// TIA Portal V19 export
FUNCTION "@LOAD CALCULATE" : Void   // FC20, LAD
{ S7_Optimized_Access := 'TRUE' }
// stored: SetENOAutomatically false
   VAR_INPUT
      "MFG PROCESS BUFF" : Int;
      "MATERIAL SUCTION BUFF" : Int;
      "MOVE PV" : Real;
      PV : Real;
   END_VAR
   VAR_OUTPUT
      "PURIFIED CALCULATE PV" : Real;
      "MATERIAL SORBITOL CALCULATE PV" : Real;
      "MATERIAL GLUCOSE CALCULATE PV" : Real;
      "MATERIAL SUCTION CALCULATE PV" : Real;
   END_VAR
BEGIN

REGION Network 1
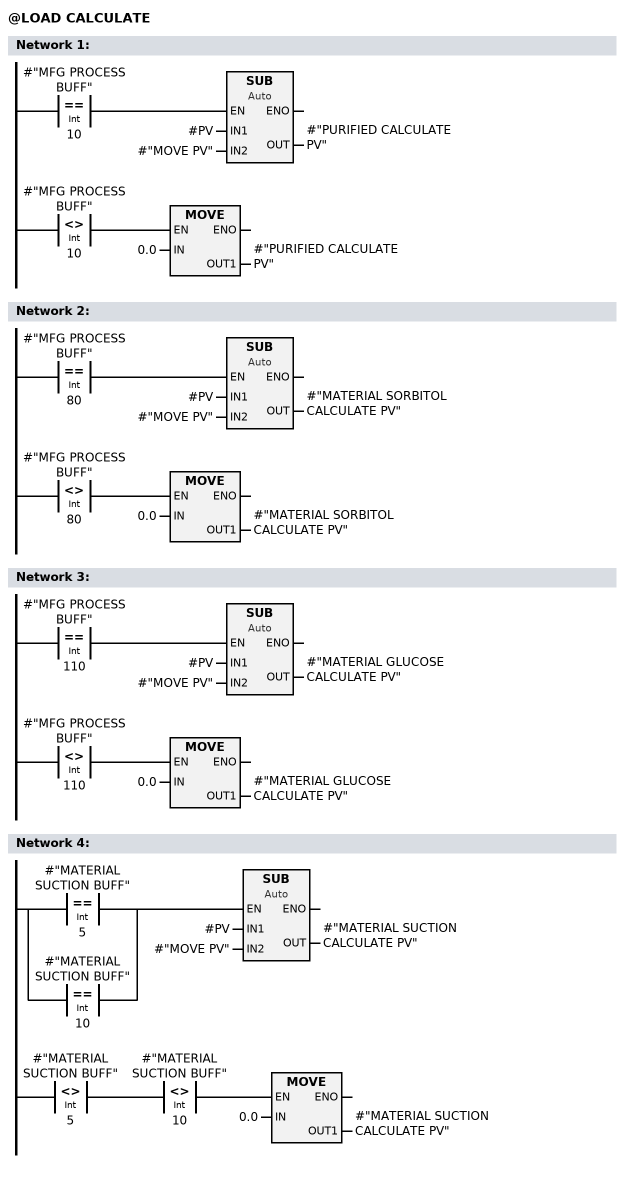
   RUNG wire#powerrail
      { S7_Templates := "SrcType := Int" } EQ_Contact(in1 := #"MFG PROCESS BUFF", in2 := 10)
      Sub(in1 := #PV, in2 := #"MOVE PV", out => #"PURIFIED CALCULATE PV")
   END_RUNG
   RUNG wire#powerrail
      { S7_Templates := "SrcType := Int" } NE_Contact(in1 := #"MFG PROCESS BUFF", in2 := 10)
      Move(in := 0.0, out1 => #"PURIFIED CALCULATE PV")
   END_RUNG
   // the same network as SCL:
   IF #"MFG PROCESS BUFF" = 10 THEN #"PURIFIED CALCULATE PV" := #PV - #"MOVE PV"; END_IF;
   IF #"MFG PROCESS BUFF" <> 10 THEN #"PURIFIED CALCULATE PV" := 0.0; END_IF;
END_REGION

REGION Network 2
   RUNG wire#powerrail
      { S7_Templates := "SrcType := Int" } EQ_Contact(in1 := #"MFG PROCESS BUFF", in2 := 80)
      Sub(in1 := #PV, in2 := #"MOVE PV", out => #"MATERIAL SORBITOL CALCULATE PV")
   END_RUNG
   RUNG wire#powerrail
      { S7_Templates := "SrcType := Int" } NE_Contact(in1 := #"MFG PROCESS BUFF", in2 := 80)
      Move(in := 0.0, out1 => #"MATERIAL SORBITOL CALCULATE PV")
   END_RUNG
   // the same network as SCL:
   IF #"MFG PROCESS BUFF" = 80 THEN #"MATERIAL SORBITOL CALCULATE PV" := #PV - #"MOVE PV"; END_IF;
   IF #"MFG PROCESS BUFF" <> 80 THEN #"MATERIAL SORBITOL CALCULATE PV" := 0.0; END_IF;
END_REGION

REGION Network 3
   RUNG wire#powerrail
      { S7_Templates := "SrcType := Int" } EQ_Contact(in1 := #"MFG PROCESS BUFF", in2 := 110)
      Sub(in1 := #PV, in2 := #"MOVE PV", out => #"MATERIAL GLUCOSE CALCULATE PV")
   END_RUNG
   RUNG wire#powerrail
      { S7_Templates := "SrcType := Int" } NE_Contact(in1 := #"MFG PROCESS BUFF", in2 := 110)
      Move(in := 0.0, out1 => #"MATERIAL GLUCOSE CALCULATE PV")
   END_RUNG
   // the same network as SCL:
   IF #"MFG PROCESS BUFF" = 110 THEN #"MATERIAL GLUCOSE CALCULATE PV" := #PV - #"MOVE PV"; END_IF;
   IF #"MFG PROCESS BUFF" <> 110 THEN #"MATERIAL GLUCOSE CALCULATE PV" := 0.0; END_IF;
END_REGION

REGION Network 4
   RUNG wire#powerrail
      { S7_Templates := "SrcType := Int" } EQ_Contact(in1 := #"MATERIAL SUCTION BUFF", in2 := 5)
      wire#w1
      Sub(in1 := #PV, in2 := #"MOVE PV", out => #"MATERIAL SUCTION CALCULATE PV")
   END_RUNG
   RUNG wire#powerrail
      { S7_Templates := "SrcType := Int" } EQ_Contact(in1 := #"MATERIAL SUCTION BUFF", in2 := 10)
   END_RUNG wire#w1
   RUNG wire#powerrail
      { S7_Templates := "SrcType := Int" } NE_Contact(in1 := #"MATERIAL SUCTION BUFF", in2 := 5)
      { S7_Templates := "SrcType := Int" } NE_Contact(in1 := #"MATERIAL SUCTION BUFF", in2 := 10)
      Move(in := 0.0, out1 => #"MATERIAL SUCTION CALCULATE PV")
   END_RUNG
   // the same network as SCL:
   IF (#"MATERIAL SUCTION BUFF" = 5) OR (#"MATERIAL SUCTION BUFF" = 10) THEN
       #"MATERIAL SUCTION CALCULATE PV" := #PV - #"MOVE PV";
   END_IF;
   IF (#"MATERIAL SUCTION BUFF" <> 5) AND (#"MATERIAL SUCTION BUFF" <> 10) THEN
       #"MATERIAL SUCTION CALCULATE PV" := 0.0;
   END_IF;
END_REGION
END_FUNCTION
